// TIA Portal project "FillerMachine" (V15)
// Maquina llenadora Fuente Pura CCN

(* hardware
DEVICE "ET 200SP station_1"  ET 200SP-Station
   slot 0: "Rack_0"  Rack  6ES5 710-8MAx1
   slot 1: "PLC_1"  CPU 1510SP-1 PN  6ES7 510-1DJ01-0AB0  V2.5
   slot 2: "DI 8x24VDC ST_1"  DI 8x24VDC ST  6ES7 131-6BF00-0BA0  V1.1
      slot 1: "DI 8x24VDC ST_1"  DI 8x24VDC ST
   slot 3: "DI 8x24VDC ST_2"  DI 8x24VDC ST  6ES7 131-6BF01-0BA0  V0.0
      slot 1: "DI 8x24VDC ST_2"  DI 8x24VDC ST
   slot 4: "DI 8x24VDC ST_3"  DI 8x24VDC ST  6ES7 131-6BF01-0BA0  V0.0
      slot 1: "DI 8x24VDC ST_3"  DI 8x24VDC ST
   slot 5: "DQ 8x24VDC/0.5A ST_1"  DQ 8x24VDC/0.5A ST  6ES7 132-6BF01-0BA0  V0.0
      slot 1: "DQ 8x24VDC/0.5A ST_1"  DQ 8x24VDC/0.5A ST
   slot 6: "DQ 8x24VDC/0.5A ST_2"  DQ 8x24VDC/0.5A ST  6ES7 132-6BF01-0BA0  V0.0
      slot 1: "DQ 8x24VDC/0.5A ST_2"  DQ 8x24VDC/0.5A ST
   slot 7: "DQ 8x24VDC/0.5A ST_3"  DQ 8x24VDC/0.5A ST  6ES7 132-6BF01-0BA0  V0.0
      slot 1: "DQ 8x24VDC/0.5A ST_3"  DQ 8x24VDC/0.5A ST
   slot 8: "Server module_1"  Server module  6ES7 193-6PA00-0AA0  V1.1
      slot 1: "Server module_1"  Server module
   slot 127: "BA 2xRJ45"  BA 2xRJ45  6ES7 193-6AR00-0AA0  V0.0
      slot 32769: "Port_1"  6ES7 193-6AR00-0AA0
      slot 32770: "Port_2"  6ES7 193-6AR00-0AA0
DEVICE "HMI_1"  KTP600 Basic color PN
   slot 0: "HMI_1"  KTP600 Basic color PN  6AV6 647-0AD11-3AX0  12.0.0.0
   slot 1: "HMI_RT_2"  KTP600 Basic color PN  6AV6 647-0AD11-3AX0  12.0.0.0
   slot 5: "HMI_1.IE_CP_1"  PROFINET Interface  12.0.0.0
      slot 1: "PROFINET Interface_1"  PROFINET Interface
         slot 1: "Port_1"  Port
*)

// ===== PLC "PLC_1"  CPU 1510SP-1 PN =====

VAR_GLOBAL   // PLC tag table "Default tag table"
   "Stop_bitin" AT %I2.2 : Bool;
   "TriggerPump" AT %I0.1 : Bool;
   "ACKPump" AT %I0.2 : Bool;
   "TriggerClamp" AT %I0.3 : Bool;
   "ACKClamp" AT %I0.4 : Bool;
   "TriggerTransp1" AT %I0.5 : Bool;
   "ACKTransp1" AT %I0.6 : Bool;
   "TriggerTransp2" AT %I0.7 : Bool;
   "ACKTransp2" AT %I1.0 : Bool;
   "SensorTransIN2" AT %I1.1 : Bool;
   "SensorInBottle" AT %I1.2 : Bool;
   "SensorOutBottle" AT %I1.3 : Bool;
   "SensorLastBottle" AT %I1.4 : Bool;
   "SensorStageIN1" AT %I1.5 : Bool;
   "SensorLevelH" AT %I1.6 : Bool;
   "SensorLevelL" AT %I1.7 : Bool;
   "SensorBottleClamp" AT %I2.0 : Bool;
   "SensorTranspClamp" AT %I2.1 : Bool;
   "PumpVLow" AT %Q0.0 : Bool;
   "PumpVHigh" AT %Q0.1 : Bool;
   "PumpStop" AT %Q0.2 : Bool;
   "MotorTap" AT %Q0.3 : Bool;
   "MotorTrans1" AT %Q0.4 : Bool;
   "MotorTrans2" AT %Q0.5 : Bool;
   "EVPrincip" AT %Q0.6 : Bool;
   "EVBlowCylindIN" AT %Q0.7 : Bool;
   "EVMandrilcylind" AT %Q1.6 : Bool;
   "EVCylindNeck" AT %Q1.7 : Bool;
   "EVDoorIn" AT %Q2.2 : Bool;
   "EVDoorOut" AT %Q2.3 : Bool;
   "EVClampBotNeck" AT %Q2.4 : Bool;
   "EVClampDoor" AT %Q2.5 : Bool;
   "EVSuperClamp" AT %Q2.6 : Bool;
   "EVCylindUpDown" AT %Q2.7 : Bool;
   "MStartTouch" AT %M11.0 : Bool;
   "MBandaT-On" AT %M10.1 : Bool;
   "MFillScreen" AT %M10.2 : Bool;
   "MBottleProcess" AT %MD100 : DInt;
   "MBottleCounterIN" AT %MD4 : DInt;
   "MBottleCounterOut" AT %MD12 : DInt;
   "MEnableClampValve" AT %MD16 : DInt;
   "MFillFinish" AT %M10.3 : Bool;
   "M_stop_bit" AT %M11.1 : Bool;
   "F_TriggerPump" AT %M11.3 : Bool;
   "F_ACKPump" AT %M11.4 : Bool;
   "F_TriggerClamp" AT %M11.5 : Bool;
   "F_ACKClamp" AT %M11.6 : Bool;
   "F_TriggerTransp1" AT %M11.7 : Bool;
   "F_ACKTransp1" AT %M20.0 : Bool;
   "F_TriggerTransp2" AT %M20.1 : Bool;
   "F_ACKTransp2" AT %M20.2 : Bool;
   "SensorTransIN2_bit" AT %M20.3 : Bool;
   "SensorInBottle_bit" AT %M20.4 : Bool;
   "SensorOutBottle_bit" AT %M20.5 : Bool;
   "SensorLastBottle_bit" AT %M20.6 : Bool;
   "SensorStageIN1_bit" AT %M20.7 : Bool;
   "SensorLevelH_bit" AT %M21.0 : Bool;
   "SensorLevelL_bit" AT %M21.1 : Bool;
   "SensorBottleClamp_bit" AT %M21.2 : Bool;
   "SensorTranspClamp_bit" AT %M21.3 : Bool;
   "PumpVLow_bit" AT %M21.4 : Bool;
   "PumpVHigh_bit" AT %M21.5 : Bool;
   "PumpStop_bit" AT %M21.6 : Bool;
   "MotorTap_bit" AT %M21.7 : Bool;
   "MotorTrans1_bit" AT %M22.0 : Bool;
   "MotorTrans2_bit" AT %M22.1 : Bool;
   "EVPrincip_bit" AT %M22.2 : Bool;
   "EVBlowCylindIN_bit" AT %M22.3 : Bool;
   "EVMandrilcylind_bit" AT %M22.4 : Bool;
   "EVCylindNeck_bit" AT %M22.5 : Bool;
   "EVDoorIn_bit" AT %M22.6 : Bool;
   "EVDoorOut_bit" AT %M22.7 : Bool;
   "EVClampBotNeck_bit" AT %M23.0 : Bool;
   "EVClampDoor_bit" AT %M23.1 : Bool;
   "EVSuperClamp_bit" AT %M23.2 : Bool;
   "Alarm" AT %M24.0 : Bool;
   "F_TriggerPump_bit" AT %M24.1 : Bool;
   "F_ACKPump_bit" AT %M24.2 : Bool;
   "F_TriggerClamp_bit" AT %M24.3 : Bool;
   "F_ACKClamp_bit" AT %M24.4 : Bool;
   "F_TriggerTransp1_bit" AT %M24.5 : Bool;
   "F_ACKTransp1_bit" AT %M24.6 : Bool;
   "F_TriggerTransp2_bit" AT %M24.7 : Bool;
   "F_ACKTransp2_bit" AT %M25.0 : Bool;
   "Run" AT %M25.1 : Bool;
   "Stop_bit" AT %M25.2 : Bool;
   "Stage0" AT %M25.3 : Bool;
   "Stage1" AT %M25.4 : Bool;
   "MBottleCounterR" AT %M25.5 : Bool;
   "MBottleProcessR" AT %M25.6 : Bool;
   "Stage2" AT %M25.7 : Bool;
   "MBottleclampRt" AT %M27.3 : Bool;
   "MBottleClamProcess" AT %MD101 : DInt;
   "MTrans1_touch" AT %M27.4 : Bool;
   "MTrans2_touch" AT %M27.5 : Bool;
   "MPump_touch" AT %M27.6 : Bool;
   "MClamp_touch" AT %M27.7 : Bool;
END_VAR

DATA_BLOCK "DB_Alarms"   // DB13
{ S7_Optimized_Access := 'FALSE' }
VERSION : 0.1
   VAR
      Stop_alm : Bool;
      T_Pump_alm : Bool;
      T_Transp1_alm : Bool;
      T_Transp2_alm : Bool;
      T_Clamp_alm_1 : Bool;
      alarms_active : Bool;
   END_VAR
BEGIN
END_DATA_BLOCK

// folder: System blocks/Program resources

DATA_BLOCK "IEC_Counter_0_DB"   // DB1
{ S7_Optimized_Access := 'TRUE' }
AUTHOR : Simatic
FAMILY : IEC
NAME : CNTR
VERSION : 1.0
// stored: InstanceOfName IEC_COUNTER
"IEC_COUNTER"
BEGIN
END_DATA_BLOCK

DATA_BLOCK "IEC_Timer_0_DB"   // DB2
{ S7_Optimized_Access := 'TRUE' }
AUTHOR : Simatic
FAMILY : IEC
NAME : IEC_TMR
VERSION : 1.0
// stored: InstanceOfName IEC_TIMER
"IEC_TIMER"
BEGIN
END_DATA_BLOCK

DATA_BLOCK "IEC_Timer_0_DB_1"   // DB3
{ S7_Optimized_Access := 'TRUE' }
AUTHOR : Simatic
FAMILY : IEC
NAME : IEC_TMR
VERSION : 1.0
// stored: InstanceOfName IEC_TIMER
"IEC_TIMER"
BEGIN
END_DATA_BLOCK

DATA_BLOCK "IEC_Timer_0_DB_3"   // DB4
{ S7_Optimized_Access := 'TRUE' }
AUTHOR : Simatic
FAMILY : IEC
NAME : IEC_TMR
VERSION : 1.0
// stored: InstanceOfName IEC_TIMER
"IEC_TIMER"
BEGIN
END_DATA_BLOCK

DATA_BLOCK "IEC_Timer_0_DB_2"   // DB5
{ S7_Optimized_Access := 'TRUE' }
AUTHOR : Simatic
FAMILY : IEC
NAME : IEC_TMR
VERSION : 1.0
// stored: InstanceOfName IEC_TIMER
"IEC_TIMER"
BEGIN
END_DATA_BLOCK

DATA_BLOCK "IEC_Timer_0_DB_4"   // DB6
{ S7_Optimized_Access := 'TRUE' }
AUTHOR : Simatic
FAMILY : IEC
NAME : IEC_TMR
VERSION : 1.0
// stored: InstanceOfName IEC_TIMER
"IEC_TIMER"
BEGIN
END_DATA_BLOCK

DATA_BLOCK "IEC_Timer_0_DB_6"   // DB8
{ S7_Optimized_Access := 'TRUE' }
AUTHOR : Simatic
FAMILY : IEC
NAME : IEC_TMR
VERSION : 1.0
// stored: InstanceOfName IEC_TIMER
"IEC_TIMER"
BEGIN
END_DATA_BLOCK

// folder: (top level)

ORGANIZATION_BLOCK "Main"   // OB1, LAD, ProgramCycle
TITLE = "Main Program Sweep (Cycle)"
{ S7_Optimized_Access := 'TRUE' }
VERSION : 0.1
   VAR_INPUT
      Initial_Call : Bool;   // Initial call of this OB
      Remanence : Bool;   // =True, if remanent data are available
   END_VAR
   VAR_TEMP   // added for the SCL form of the ladder/FBD networks
      _w1 : Bool;
      _w2 : Bool;
   END_VAR
BEGIN

REGION Network 1
   // Start  Stop Control
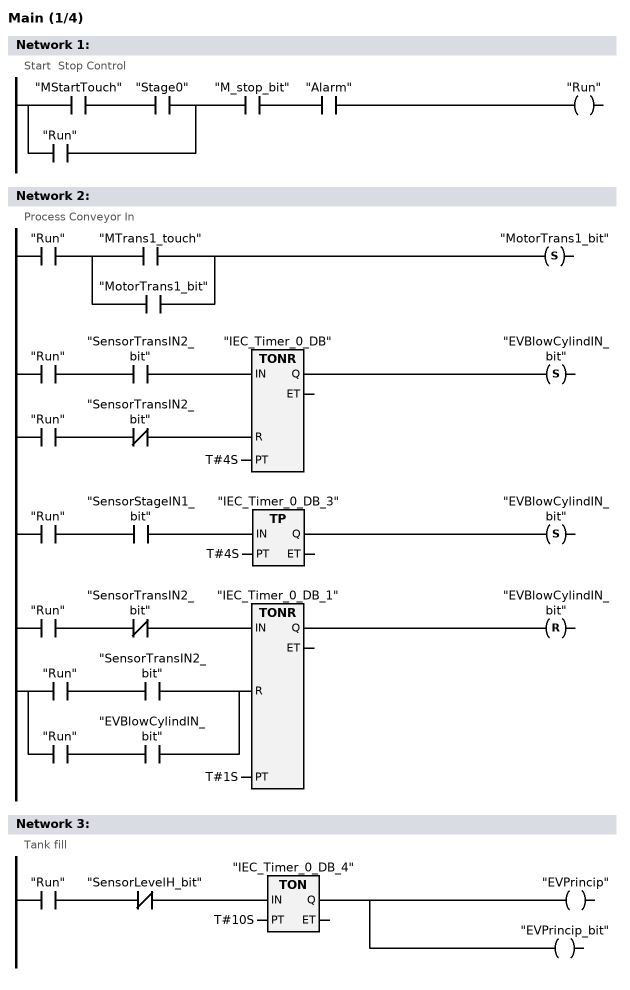
   RUNG wire#powerrail
      Contact( "MStartTouch" )
      Contact( "Stage0" )
      wire#w1
      Contact( "M_stop_bit" )
      Contact( "Alarm" )
      Coil( "Run" )
   END_RUNG
   RUNG wire#powerrail
      Contact( "Run" )
   END_RUNG wire#w1
   // the same network as SCL:
   "Run" := (("MStartTouch" AND "Stage0") OR "Run") AND "M_stop_bit" AND "Alarm";
END_REGION

REGION Network 2
   // Process Conveyor In
   IF "Run" AND ("MTrans1_touch" OR "MotorTrans1_bit") THEN "MotorTrans1_bit" := TRUE; END_IF;
   "IEC_Timer_0_DB".TONR(IN := "Run" AND "SensorTransIN2_bit",
                         R := "Run" AND NOT "SensorTransIN2_bit",
                         PT := T#4S);
   IF "IEC_Timer_0_DB".Q THEN "EVBlowCylindIN_bit" := TRUE; END_IF;
   "IEC_Timer_0_DB_3".TP(IN := "Run" AND "SensorStageIN1_bit", PT := T#4S);
   IF "IEC_Timer_0_DB_3".Q THEN "EVBlowCylindIN_bit" := TRUE; END_IF;
   "IEC_Timer_0_DB_1".TONR(IN := "Run" AND NOT "SensorTransIN2_bit",
                           R := ("Run" AND "SensorTransIN2_bit") OR ("Run" AND "EVBlowCylindIN_bit"),
                           PT := T#1S);
   IF "IEC_Timer_0_DB_1".Q THEN "EVBlowCylindIN_bit" := FALSE; END_IF;
END_REGION

REGION Network 3
   // Tank fill
   "IEC_Timer_0_DB_4".TON(IN := "Run" AND NOT "SensorLevelH_bit", PT := T#10S);
   "EVPrincip" := "IEC_Timer_0_DB_4".Q;
   "EVPrincip_bit" := "IEC_Timer_0_DB_4".Q;
END_REGION

REGION Network 4
   // Process Filling Bottle
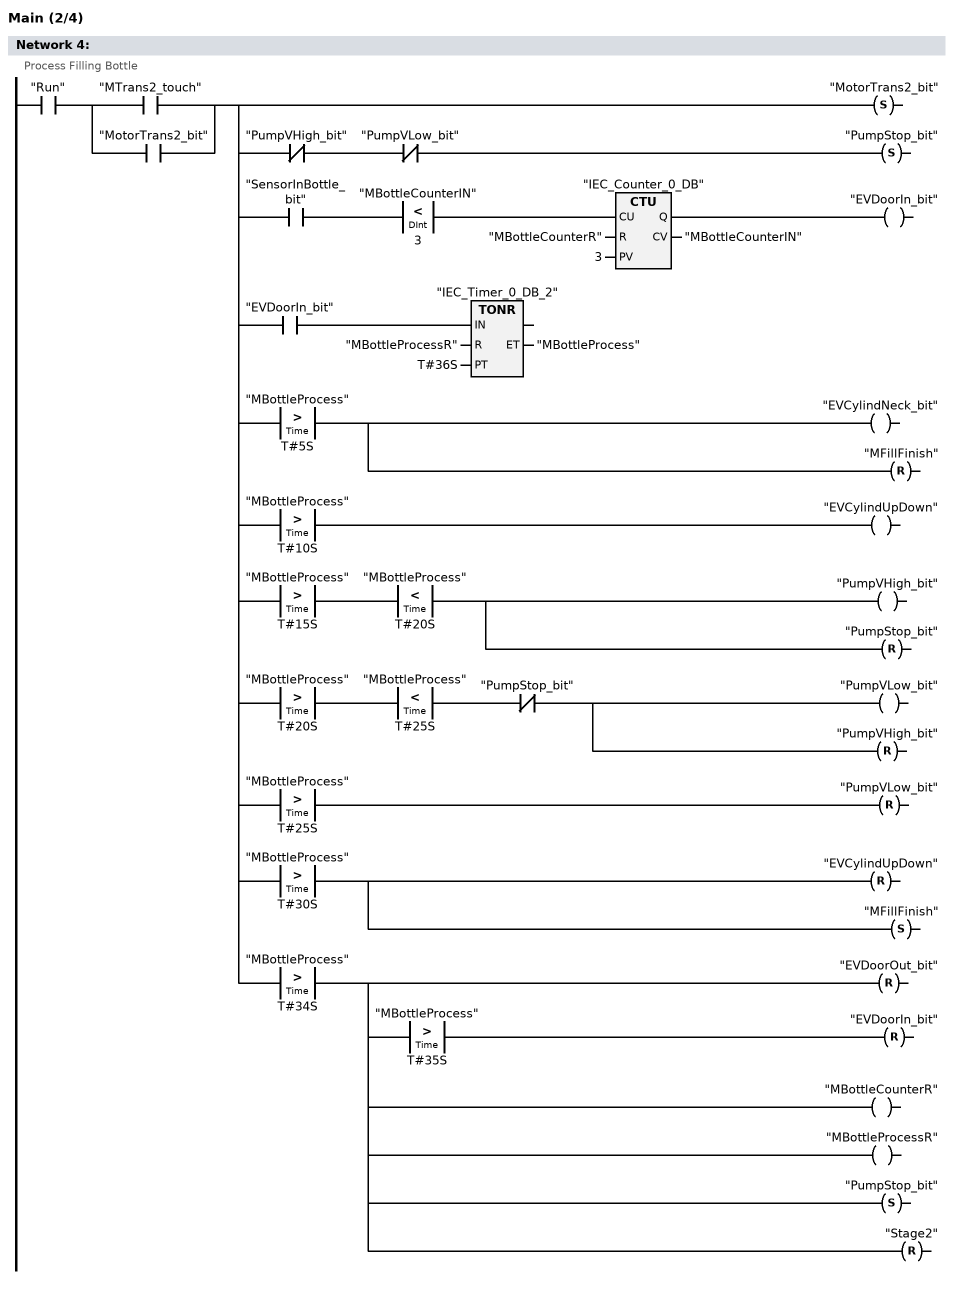
   #_w1 := "Run" AND ("MTrans2_touch" OR "MotorTrans2_bit");
   IF #_w1 THEN "MotorTrans2_bit" := TRUE; END_IF;
   IF #_w1 AND NOT "PumpVHigh_bit" AND NOT "PumpVLow_bit" THEN "PumpStop_bit" := TRUE; END_IF;
   "IEC_Counter_0_DB".CTU(CU := #_w1 AND "SensorInBottle_bit" AND ("MBottleCounterIN" < 3),
                          R := "MBottleCounterR",
                          PV := 3,
                          CV => "MBottleCounterIN");
   "EVDoorIn_bit" := "IEC_Counter_0_DB".Q;
   "IEC_Timer_0_DB_2".TONR(IN := #_w1 AND "EVDoorIn_bit",
                           R := "MBottleProcessR",
                           PT := T#36S,
                           ET => "MBottleProcess");
   "EVCylindNeck_bit" := #_w1 AND ("MBottleProcess" > T#5S);
   IF "EVCylindNeck_bit" THEN "MFillFinish" := FALSE; END_IF;
   "EVCylindUpDown" := #_w1 AND ("MBottleProcess" > T#10S);
   "PumpVHigh_bit" := #_w1 AND ("MBottleProcess" > T#15S) AND ("MBottleProcess" < T#20S);
   IF "PumpVHigh_bit" THEN "PumpStop_bit" := FALSE; END_IF;
   "PumpVLow_bit" := #_w1 AND ("MBottleProcess" > T#20S) AND ("MBottleProcess" < T#25S) AND NOT "PumpStop_bit";
   IF "PumpVLow_bit" THEN "PumpVHigh_bit" := FALSE; END_IF;
   IF #_w1 AND ("MBottleProcess" > T#25S) THEN "PumpVLow_bit" := FALSE; END_IF;
   IF #_w1 AND ("MBottleProcess" > T#30S) THEN
       "EVCylindUpDown" := FALSE;
       "MFillFinish" := TRUE;
   END_IF;
   #_w2 := #_w1 AND ("MBottleProcess" > T#34S);
   IF #_w2 THEN "EVDoorOut_bit" := FALSE; END_IF;
   IF #_w2 AND ("MBottleProcess" > T#35S) THEN "EVDoorIn_bit" := FALSE; END_IF;
   "MBottleCounterR" := #_w2;
   "MBottleProcessR" := #_w2;
   IF #_w2 THEN
       "PumpStop_bit" := TRUE;
       "Stage2" := FALSE;
   END_IF;
END_REGION

REGION Network 5
   // Cylin dre out
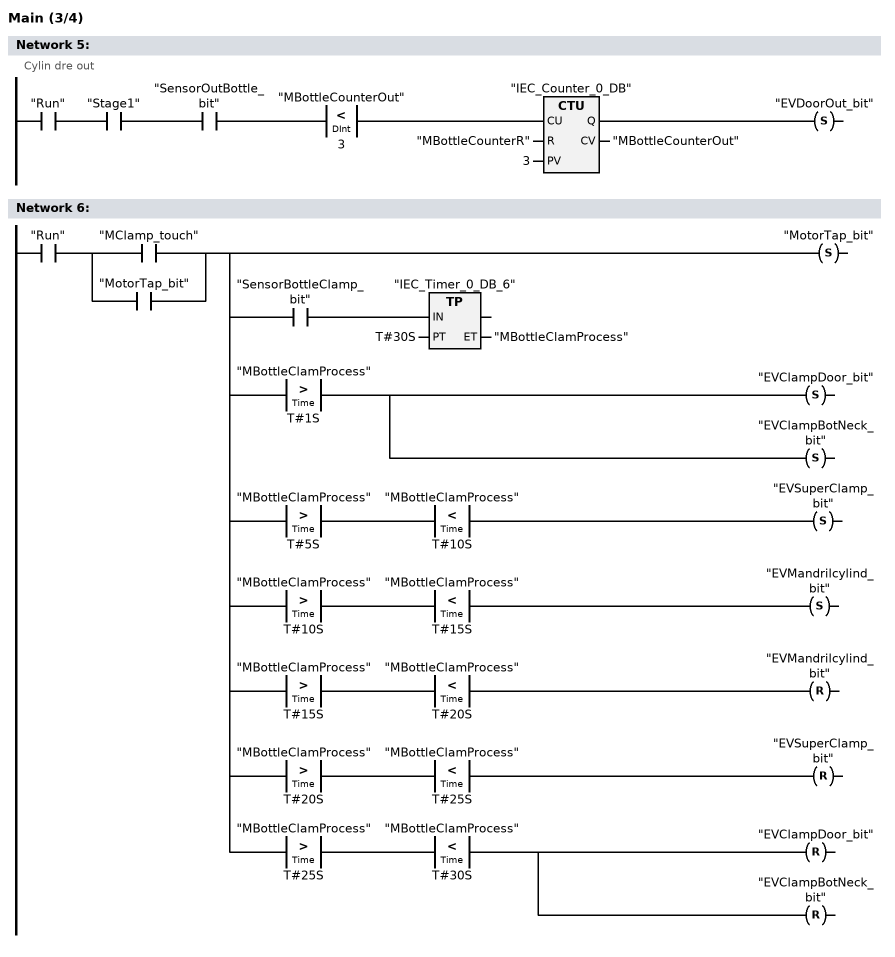
   "IEC_Counter_0_DB".CTU(CU := "Run" AND "Stage1" AND "SensorOutBottle_bit" AND ("MBottleCounterOut" < 3),
                          R := "MBottleCounterR",
                          PV := 3,
                          CV => "MBottleCounterOut");
   IF "IEC_Counter_0_DB".Q THEN "EVDoorOut_bit" := TRUE; END_IF;
END_REGION

REGION Network 6
   #_w1 := "Run" AND ("MClamp_touch" OR "MotorTap_bit");
   IF #_w1 THEN "MotorTap_bit" := TRUE; END_IF;
   "IEC_Timer_0_DB_6".TP(IN := #_w1 AND "SensorBottleClamp_bit", PT := T#30S, ET => "MBottleClamProcess");
   IF #_w1 AND ("MBottleClamProcess" > T#1S) THEN
       "EVClampDoor_bit" := TRUE;
       "EVClampBotNeck_bit" := TRUE;
   END_IF;
   IF #_w1 AND ("MBottleClamProcess" > T#5S) AND ("MBottleClamProcess" < T#10S) THEN
       "EVSuperClamp_bit" := TRUE;
   END_IF;
   IF #_w1 AND ("MBottleClamProcess" > T#10S) AND ("MBottleClamProcess" < T#15S) THEN
       "EVMandrilcylind_bit" := TRUE;
   END_IF;
   IF #_w1 AND ("MBottleClamProcess" > T#15S) AND ("MBottleClamProcess" < T#20S) THEN
       "EVMandrilcylind_bit" := FALSE;
   END_IF;
   IF #_w1 AND ("MBottleClamProcess" > T#20S) AND ("MBottleClamProcess" < T#25S) THEN
       "EVSuperClamp_bit" := FALSE;
   END_IF;
   IF #_w1 AND ("MBottleClamProcess" > T#25S) AND ("MBottleClamProcess" < T#30S) THEN
       "EVClampDoor_bit" := FALSE;
       "EVClampBotNeck_bit" := FALSE;
   END_IF;
END_REGION

REGION Network 7
   // Minor bits
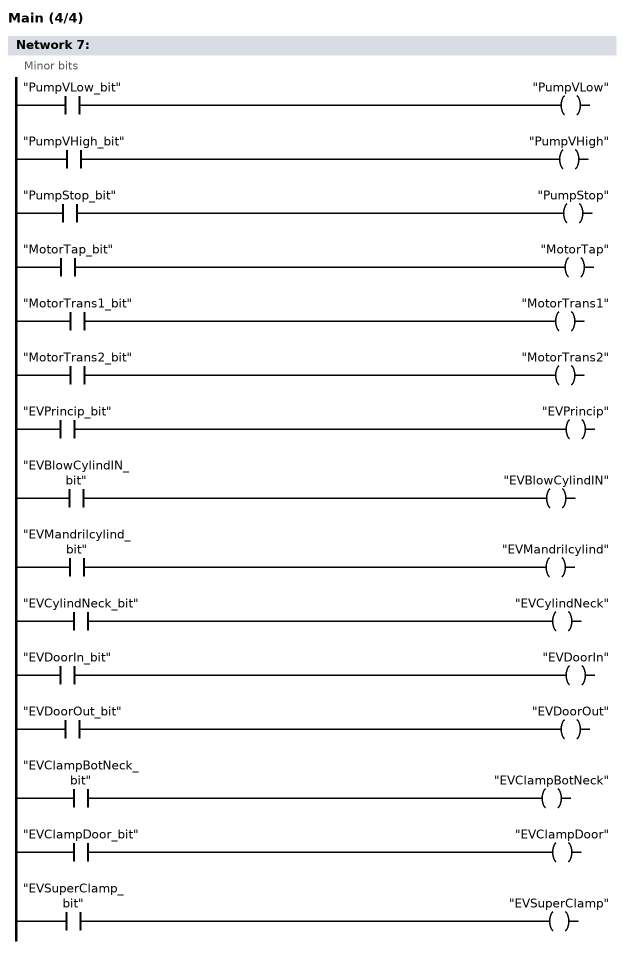
   RUNG wire#powerrail
      Contact( "PumpVLow_bit" )
      Coil( "PumpVLow" )
   END_RUNG
   RUNG wire#powerrail
      Contact( "PumpVHigh_bit" )
      Coil( "PumpVHigh" )
   END_RUNG
   RUNG wire#powerrail
      Contact( "PumpStop_bit" )
      Coil( "PumpStop" )
   END_RUNG
   RUNG wire#powerrail
      Contact( "MotorTap_bit" )
      Coil( "MotorTap" )
   END_RUNG
   RUNG wire#powerrail
      Contact( "MotorTrans1_bit" )
      Coil( "MotorTrans1" )
   END_RUNG
   RUNG wire#powerrail
      Contact( "MotorTrans2_bit" )
      Coil( "MotorTrans2" )
   END_RUNG
   RUNG wire#powerrail
      Contact( "EVPrincip_bit" )
      Coil( "EVPrincip" )
   END_RUNG
   RUNG wire#powerrail
      Contact( "EVBlowCylindIN_bit" )
      Coil( "EVBlowCylindIN" )
   END_RUNG
   RUNG wire#powerrail
      Contact( "EVMandrilcylind_bit" )
      Coil( "EVMandrilcylind" )
   END_RUNG
   RUNG wire#powerrail
      Contact( "EVCylindNeck_bit" )
      Coil( "EVCylindNeck" )
   END_RUNG
   RUNG wire#powerrail
      Contact( "EVDoorIn_bit" )
      Coil( "EVDoorIn" )
   END_RUNG
   RUNG wire#powerrail
      Contact( "EVDoorOut_bit" )
      Coil( "EVDoorOut" )
   END_RUNG
   RUNG wire#powerrail
      Contact( "EVClampBotNeck_bit" )
      Coil( "EVClampBotNeck" )
   END_RUNG
   RUNG wire#powerrail
      Contact( "EVClampDoor_bit" )
      Coil( "EVClampDoor" )
   END_RUNG
   RUNG wire#powerrail
      Contact( "EVSuperClamp_bit" )
      Coil( "EVSuperClamp" )
   END_RUNG
   // the same network as SCL:
   "PumpVLow" := "PumpVLow_bit";
   "PumpVHigh" := "PumpVHigh_bit";
   "PumpStop" := "PumpStop_bit";
   "MotorTap" := "MotorTap_bit";
   "MotorTrans1" := "MotorTrans1_bit";
   "MotorTrans2" := "MotorTrans2_bit";
   "EVPrincip" := "EVPrincip_bit";
   "EVBlowCylindIN" := "EVBlowCylindIN_bit";
   "EVMandrilcylind" := "EVMandrilcylind_bit";
   "EVCylindNeck" := "EVCylindNeck_bit";
   "EVDoorIn" := "EVDoorIn_bit";
   "EVDoorOut" := "EVDoorOut_bit";
   "EVClampBotNeck" := "EVClampBotNeck_bit";
   "EVClampDoor" := "EVClampDoor_bit";
   "EVSuperClamp" := "EVSuperClamp_bit";
END_REGION
END_ORGANIZATION_BLOCK

ORGANIZATION_BLOCK "Alarms_block"   // OB123, LAD, ProgramCycle
TITLE = "Main Program Sweep (Cycle)"
{ S7_Optimized_Access := 'TRUE' }
VERSION : 0.1
   VAR_INPUT
      Initial_Call : Bool;   // Initial call of this OB
      Remanence : Bool;   // =True, if remanent data are available
   END_VAR
BEGIN

REGION Network 1
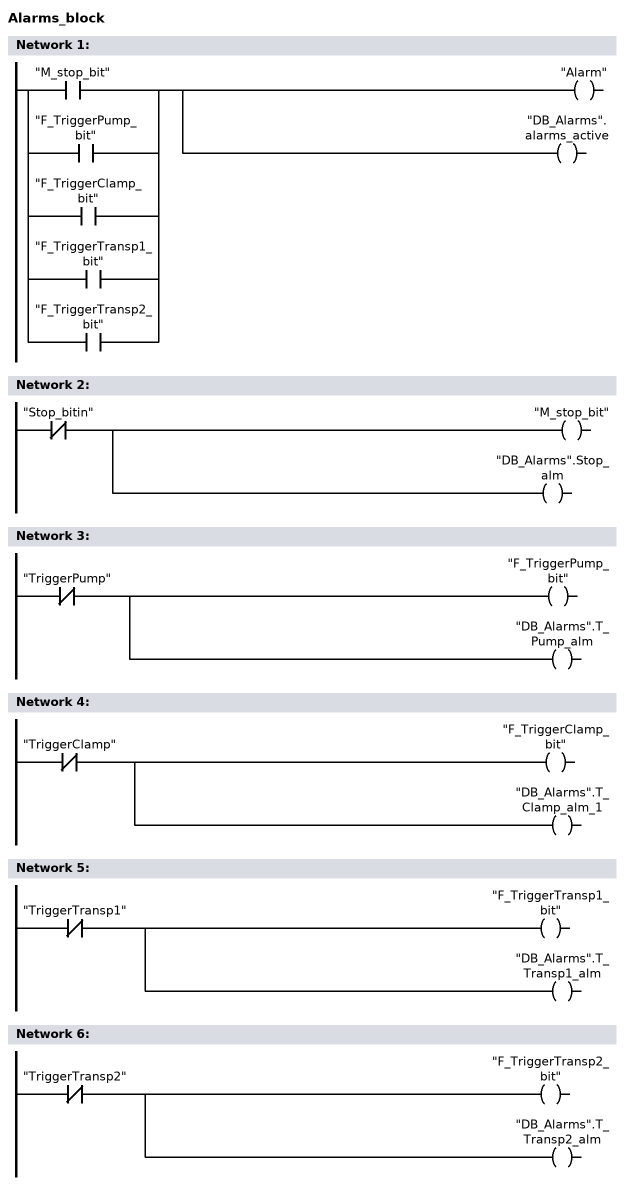
   RUNG wire#powerrail
      Contact( "M_stop_bit" )
      wire#w1
      Coil( "Alarm" )
   END_RUNG
   RUNG wire#powerrail
      Contact( "F_TriggerPump_bit" )
   END_RUNG wire#w1
   RUNG wire#powerrail
      Contact( "F_TriggerClamp_bit" )
   END_RUNG wire#w1
   RUNG wire#powerrail
      Contact( "F_TriggerTransp1_bit" )
   END_RUNG wire#w1
   RUNG wire#powerrail
      Contact( "F_TriggerTransp2_bit" )
   END_RUNG wire#w1
   RUNG wire#w1
      Coil( "DB_Alarms".alarms_active )
   END_RUNG
   // the same network as SCL:
   "Alarm" := "M_stop_bit" OR "F_TriggerPump_bit" OR "F_TriggerClamp_bit" OR "F_TriggerTransp1_bit" OR "F_TriggerTransp2_bit";
   "DB_Alarms".alarms_active := "Alarm";
END_REGION

REGION Network 2
   RUNG wire#powerrail
      I_Contact( "Stop_bitin" )
      wire#w1
      Coil( "M_stop_bit" )
   END_RUNG
   RUNG wire#w1
      Coil( "DB_Alarms".Stop_alm )
   END_RUNG
   // the same network as SCL:
   "M_stop_bit" := NOT "Stop_bitin";
   "DB_Alarms".Stop_alm := NOT "Stop_bitin";
END_REGION

REGION Network 3
   RUNG wire#powerrail
      I_Contact( "TriggerPump" )
      wire#w1
      Coil( "F_TriggerPump_bit" )
   END_RUNG
   RUNG wire#w1
      Coil( "DB_Alarms".T_Pump_alm )
   END_RUNG
   // the same network as SCL:
   "F_TriggerPump_bit" := NOT "TriggerPump";
   "DB_Alarms".T_Pump_alm := NOT "TriggerPump";
END_REGION

REGION Network 4
   RUNG wire#powerrail
      I_Contact( "TriggerClamp" )
      wire#w1
      Coil( "F_TriggerClamp_bit" )
   END_RUNG
   RUNG wire#w1
      Coil( "DB_Alarms".T_Clamp_alm_1 )
   END_RUNG
   // the same network as SCL:
   "F_TriggerClamp_bit" := NOT "TriggerClamp";
   "DB_Alarms".T_Clamp_alm_1 := NOT "TriggerClamp";
END_REGION

REGION Network 5
   RUNG wire#powerrail
      I_Contact( "TriggerTransp1" )
      wire#w1
      Coil( "F_TriggerTransp1_bit" )
   END_RUNG
   RUNG wire#w1
      Coil( "DB_Alarms".T_Transp1_alm )
   END_RUNG
   // the same network as SCL:
   "F_TriggerTransp1_bit" := NOT "TriggerTransp1";
   "DB_Alarms".T_Transp1_alm := NOT "TriggerTransp1";
END_REGION

REGION Network 6
   RUNG wire#powerrail
      I_Contact( "TriggerTransp2" )
      wire#w1
      Coil( "F_TriggerTransp2_bit" )
   END_RUNG
   RUNG wire#w1
      Coil( "DB_Alarms".T_Transp2_alm )
   END_RUNG
   // the same network as SCL:
   "F_TriggerTransp2_bit" := NOT "TriggerTransp2";
   "DB_Alarms".T_Transp2_alm := NOT "TriggerTransp2";
END_REGION
END_ORGANIZATION_BLOCK

ORGANIZATION_BLOCK "Stages"   // OB124, LAD, ProgramCycle
TITLE = "Main Program Sweep (Cycle)"
{ S7_Optimized_Access := 'TRUE' }
VERSION : 0.1
   VAR_INPUT
      Initial_Call : Bool;   // Initial call of this OB
      Remanence : Bool;   // =True, if remanent data are available
   END_VAR
   VAR_TEMP   // added for the SCL form of the ladder/FBD networks
      _w1 : Bool;
   END_VAR
BEGIN

REGION Network 1
   // Stage0
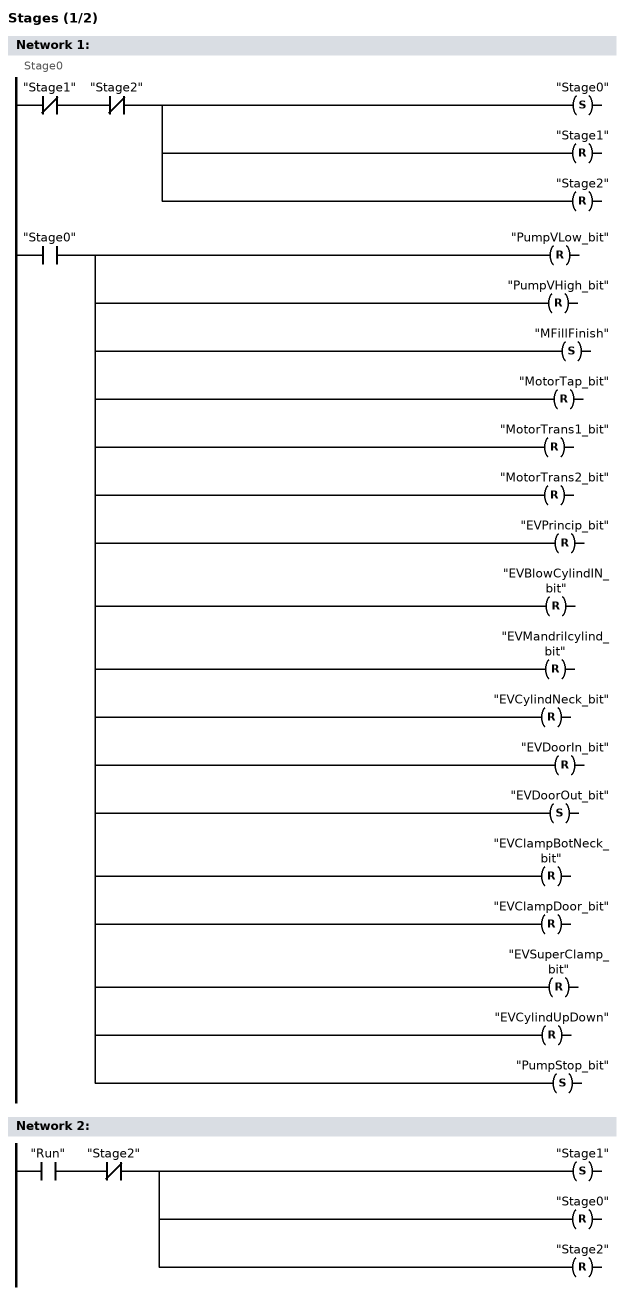
   RUNG wire#powerrail
      I_Contact( "Stage1" )
      I_Contact( "Stage2" )
      wire#w1
      S_Coil( "Stage0" )
   END_RUNG
   RUNG wire#w1
      R_Coil( "Stage1" )
   END_RUNG
   RUNG wire#w1
      R_Coil( "Stage2" )
   END_RUNG
   RUNG wire#powerrail
      Contact( "Stage0" )
      wire#w2
      R_Coil( "PumpVLow_bit" )
   END_RUNG
   RUNG wire#w2
      R_Coil( "PumpVHigh_bit" )
   END_RUNG
   RUNG wire#w2
      S_Coil( "MFillFinish" )
   END_RUNG
   RUNG wire#w2
      R_Coil( "MotorTap_bit" )
   END_RUNG
   RUNG wire#w2
      R_Coil( "MotorTrans1_bit" )
   END_RUNG
   RUNG wire#w2
      R_Coil( "MotorTrans2_bit" )
   END_RUNG
   RUNG wire#w2
      R_Coil( "EVPrincip_bit" )
   END_RUNG
   RUNG wire#w2
      R_Coil( "EVBlowCylindIN_bit" )
   END_RUNG
   RUNG wire#w2
      R_Coil( "EVMandrilcylind_bit" )
   END_RUNG
   RUNG wire#w2
      R_Coil( "EVCylindNeck_bit" )
   END_RUNG
   RUNG wire#w2
      R_Coil( "EVDoorIn_bit" )
   END_RUNG
   RUNG wire#w2
      S_Coil( "EVDoorOut_bit" )
   END_RUNG
   RUNG wire#w2
      R_Coil( "EVClampBotNeck_bit" )
   END_RUNG
   RUNG wire#w2
      R_Coil( "EVClampDoor_bit" )
   END_RUNG
   RUNG wire#w2
      R_Coil( "EVSuperClamp_bit" )
   END_RUNG
   RUNG wire#w2
      R_Coil( "EVCylindUpDown" )
   END_RUNG
   RUNG wire#w2
      S_Coil( "PumpStop_bit" )
   END_RUNG
   // the same network as SCL:
   IF NOT "Stage1" AND NOT "Stage2" THEN "Stage0" := TRUE; END_IF;
   #_w1 := NOT "Stage1" AND NOT "Stage2";
   IF #_w1 THEN
       "Stage1" := FALSE;
       "Stage2" := FALSE;
   END_IF;
   IF "Stage0" THEN
       "PumpVLow_bit" := FALSE;
       "PumpVHigh_bit" := FALSE;
       "MFillFinish" := TRUE;
       "MotorTap_bit" := FALSE;
       "MotorTrans1_bit" := FALSE;
       "MotorTrans2_bit" := FALSE;
       "EVPrincip_bit" := FALSE;
       "EVBlowCylindIN_bit" := FALSE;
       "EVMandrilcylind_bit" := FALSE;
       "EVCylindNeck_bit" := FALSE;
       "EVDoorIn_bit" := FALSE;
       "EVDoorOut_bit" := TRUE;
       "EVClampBotNeck_bit" := FALSE;
       "EVClampDoor_bit" := FALSE;
       "EVSuperClamp_bit" := FALSE;
       "EVCylindUpDown" := FALSE;
       "PumpStop_bit" := TRUE;
   END_IF;
END_REGION

REGION Network 2
   RUNG wire#powerrail
      Contact( "Run" )
      I_Contact( "Stage2" )
      wire#w1
      S_Coil( "Stage1" )
   END_RUNG
   RUNG wire#w1
      R_Coil( "Stage0" )
   END_RUNG
   RUNG wire#w1
      R_Coil( "Stage2" )
   END_RUNG
   // the same network as SCL:
   IF "Run" AND NOT "Stage2" THEN
       "Stage1" := TRUE;
       "Stage0" := FALSE;
       "Stage2" := FALSE;
   END_IF;
END_REGION

REGION Network 4
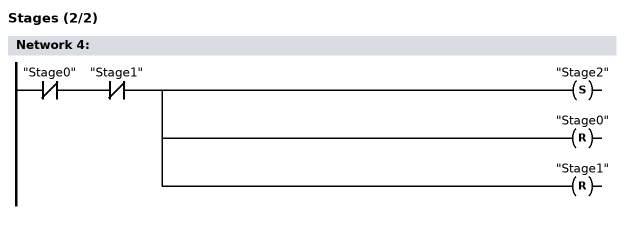
   RUNG wire#powerrail
      I_Contact( "Stage0" )
      I_Contact( "Stage1" )
      wire#w1
      S_Coil( "Stage2" )
   END_RUNG
   RUNG wire#w1
      R_Coil( "Stage0" )
   END_RUNG
   RUNG wire#w1
      R_Coil( "Stage1" )
   END_RUNG
   // the same network as SCL:
   IF NOT "Stage0" AND NOT "Stage1" THEN "Stage2" := TRUE; END_IF;
   #_w1 := NOT "Stage0" AND NOT "Stage1";
   IF #_w1 THEN
       "Stage0" := FALSE;
       "Stage1" := FALSE;
   END_IF;
END_REGION
END_ORGANIZATION_BLOCK

(* ===== HMI "HMI_RT_2" =====
system functions are stored by id; their names below are inferred from use
connection "HMI_Connection_1": ETHERNET, SMART_S7_1500_OMS

HMI tags "Default tag table"
   "HMI_Tag_1" : UInt AT %DB13.DBW0, 1 s
   "Tag_ScreenNumber" : UInt, internal
   "MStartTouch" : Bool = PLC MStartTouch AT %M11.0, 1 s
   "MTrans1_touch" : Bool = PLC MTrans1_touch AT %M27.4, 1 s
   "MTrans2_touch" : Bool = PLC MTrans2_touch AT %M27.5, 1 s
   "MClamp_touch" : Bool = PLC MClamp_touch AT %M27.7, 1 s

discrete alarms
   1: 'Alarma Paro de emergencia', class Errors, trigger "HMI_Tag_1" bit 0
   2: 'Disparo de Bomba', class Errors, trigger "HMI_Tag_1" bit 2
   3: 'Disparo del Motor Transportador 1', class Errors, trigger "HMI_Tag_1" bit 3
   4: 'Disparo del Motor Transportador 2', class Errors, trigger "HMI_Tag_1" bit 4
   5: 'Disparo del Motor Clamp', class Errors, trigger "HMI_Tag_1" bit 5
   6: 'Alarmas Activas', class Errors, trigger "HMI_Tag_1" bit 6

Template "Template_1" 320x240
   Button "Template_Button" at 266,202 size 52x37; TextOff 'Text'; PictureOff "ExitRuntime_KTP700_Basic_PN_TR"
      on Release: StopRuntime(0)
   Button "Template_Button_1" at 213,202 size 52x37; TextOff 'Text'
   Button "Template_Button_2" at 160,202 size 52x37; TextOff 'Text'
   Button "Template_Button_3" at 107,202 size 52x37; TextOff 'Text'; PictureOff "Graphic_3"
      on Release: ActivateScreen("Process", 0)
   Button "Template_Button_4" at 54,202 size 52x37; TextOff 'Text'; PictureOff "AlarmDisplay_KTP600_Basic_color_PN"
      on Release: ActivateScreen("Alarms", 0)
   Button "Alarms" at 1,202 size 52x37; TextOff 'Alarms'; PictureOn "AlarmDisplay_KTP600_Basic_color_PN"; PictureOff "Home"
      on Release: ActivateScreen("Main", 0)
   SymbolicIOField "Symbolic_IO_Field_Screen" at 69,7 size 164x24; TextOff '0'; TextOn '1'; TextList "TextList_ScreenNames"
      on Change: ActivateScreenByNumber("Tag_ScreenNumber", 0)
      ProcessValue <- "Tag_ScreenNumber"
   DateTimeField "HmiScreenItemData" at 235,19 size 85x19
   DateTimeField "HmiScreenItemData_1" at 235,0 size 85x19
   GraphicView "Logo" at 0,0 size 67x38; Picture "LogoHorizontal-e1441054646412"

screen "Main" 320x240, template "Template_1"
   on GenerateScreen: SetTag("Tag_ScreenNumber", 1)
   GraphicView "Graphic view_1" at 3,53 size 223x59; Picture "LogoHorizontal-e1441054646412"
   Button "Button_1" at 10,146 size 96x32; TextOff 'Start'
      on Press: SetBit("MStartTouch")

screen "Alarms" 320x240, template "Template_1"
   on GenerateScreen: SetTag("Tag_ScreenNumber", 2)
   AlarmView "Alarm view_1" at 0,40 size 320x141

screen "Process" 320x240, template "Template_1"
   on GenerateScreen: SetTag("Tag_ScreenNumber", 3)
   Button "Button_1" at 10,146 size 96x32; TextOff 'Bomba'
      on Press: SetBit("MStartTouch")
   Button "Button_2" at 10,102 size 96x32; TextOff 'B Trans 2'
      on Press: SetBit("MTrans2_touch")
   Button "Button_3" at 10,58 size 96x32; TextOff 'B Trans 1'
      on Press: SetBit("MTrans1_touch")
   Button "Button_4" at 124,58 size 96x32; TextOff 'Motor Tap.'
      on Press: SetBit("MClamp_touch")
*)